LIN {X 0,Y 64.411,Z 489.736,A -85,B 0,C 180,E1 -30610.877,E2 -30610.877} C_VEL
LIN {X 0,Y 51.154,Z 493.638,A -85,B 0,C 180,E1 -30615.897,E2 -30615.897} C_VEL
LIN {X 0,Y 44.77,Z 495.003,A -85,B 0,C 180,E1 -30619.623,E2 -30619.623} C_VEL
LIN {X 0,Y 33.01,Z 496.515,A -85,B 0,C 180,E1 -30631.605,E2 -30631.605} C_VEL
LIN {X 0,Y 24.283,Z 496.546,A -85,B 0,C 180,E1 -30654.624,E2 -30654.624} C_VEL
LIN {X 0,Y 22.308,Z 495.994,A -85,B 0,C 180,E1 -30671.629,E2 -30671.629} C_VEL
LIN {X 0,Y 21.842,Z 494.93,A -85,B 0,C 180,E1 -30689.992,E2 -30689.992} C_VEL
LIN {X 0,Y 22.673,Z 492.2,A -85,B 0,C 180,E1 -30717.699,E2 -30717.699} C_VEL
LIN {X 0,Y 27.806,Z 488.413,A -85,B 0,C 180,E1 -30739.3,E2 -30739.3} C_VEL
LIN {X 0,Y 35.581,Z 483.511,A -85,B 0,C 180,E1 -30752.715,E2 -30752.715} C_VEL
LIN {X 0,Y 44.643,Z 477.362,A -85,B 0,C 180,E1 -30760.815,E2 -30760.815} C_VEL
LIN {X 0,Y 54.307,Z 469.729,A -85,B 0,C 180,E1 -30766.054,E2 -30766.054} C_VEL
LIN {X 0,Y 62.602,Z 461.942,A -85,B 0,C 180,E1 -30769.19,E2 -30769.19} C_VEL
LIN {X 0,Y 71.072,Z 452.525,A -85,B 0,C 180,E1 -30771.416,E2 -30771.416} C_VEL
LIN {X 0,Y 78.787,Z 442.074,A -85,B 0,C 180,E1 -30772.895,E2 -30772.895} C_VEL
LIN {X 0,Y 85.688,Z 430.488,A -85,B 0,C 180,E1 -30773.94,E2 -30773.94} C_VEL
LIN {X 0,Y 91.281,Z 418.187,A -85,B 0,C 180,E1 -30774.899,E2 -30774.899} C_VEL
LIN {X 0,Y 95.798,Z 404.539,A -85,B 0,C 180,E1 -30775.577,E2 -30775.577} C_VEL
LIN {X 0,Y 98.056,Z 394.55,A -85,B 0,C 180,E1 -30776.019,E2 -30776.019} C_VEL
LIN {X 0,Y 99.588,Z 382.636,A -85,B 0,C 180,E1 -30777.143,E2 -30777.143} C_VEL
LIN {X 0,Y 99.215,Z 380.276,A -85,B 0,C 180,E1 -30780.904,E2 -30780.904} C_VEL
LIN {X 0,Y 99.074,Z 379.59,A -85,B 0,C 180,E1 -30784.069,E2 -30784.069} C_VEL
LIN {X 0,Y 99.228,Z 380.869,A -85,B 0,C 180,E1 -30789.529,E2 -30789.529} C_VEL
LIN {X 0,Y 99.747,Z 383.531,A -85,B 0,C 180,E1 -30793.797,E2 -30793.797} C_VEL
LIN {X 0,Y 97.367,Z 397.045,A -85,B 0,C 180,E1 -30794.611,E2 -30794.611} C_VEL
LIN {X 0,Y 93.817,Z 409.498,A -85,B 0,C 180,E1 -30795.532,E2 -30795.532} C_VEL
LIN {X 0,Y 88.903,Z 421.701,A -85,B 0,C 180,E1 -30796.731,E2 -30796.731} C_VEL
LIN {X 0,Y 82.394,Z 434,A -85,B 0,C 180,E1 -30798.4,E2 -30798.4} C_VEL
LIN {X 0,Y 75.011,Z 444.958,A -85,B 0,C 180,E1 -30800.468,E2 -30800.468} C_VEL
LIN {X 0,Y 66.865,Z 454.739,A -85,B 0,C 180,E1 -30803.129,E2 -30803.129} C_VEL
LIN {X 0,Y 57.311,Z 464.214,A -85,B 0,C 180,E1 -30807.253,E2 -30807.253} C_VEL
LIN {X 0,Y 51.041,Z 469.447,A -85,B 0,C 180,E1 -30810.706,E2 -30810.706} C_VEL
LIN {X 0,Y 46.551,Z 472.773,A -85,B 0,C 180,E1 -30812.993,E2 -30812.993} C_VEL
LIN {X 0,Y 38.26,Z 477.884,A -85,B 0,C 180,E1 -30815.633,E2 -30815.633} C_VEL
LIN {X 0,Y 29.677,Z 482.288,A -85,B 0,C 180,E1 -30819.804,E2 -30819.804} C_VEL
LIN {X 0,Y 24.982,Z 484.511,A -85,B 0,C 180,E1 -30825.843,E2 -30825.843} C_VEL
LIN {X 0,Y 18.331,Z 488.004,A -85,B 0,C 180,E1 -30847.467,E2 -30847.467} C_VEL
LIN {X 0,Y 16.306,Z 489.794,A -85,B 0,C 180,E1 -30870.01,E2 -30870.01} C_VEL
LIN {X 0,Y 17.09,Z 491.165,A -85,B 0,C 180,E1 -30894.293,E2 -30894.293} C_VEL
LIN {X 0,Y 25.119,Z 492.78,A -85,B 0,C 180,E1 -30927.083,E2 -30927.083} C_VEL
LIN {X 0,Y 36.936,Z 492.769,A -85,B 0,C 180,E1 -30942.069,E2 -30942.069} C_VEL
LIN {X 0,Y 49.983,Z 491.209,A -85,B 0,C 180,E1 -30949.828,E2 -30949.828} C_VEL
LIN {X 0,Y 59.176,Z 489.158,A -85,B 0,C 180,E1 -30953.178,E2 -30953.178} C_VEL
LIN {X 0,Y 70.438,Z 485.63,A -85,B 0,C 180,E1 -30956.175,E2 -30956.175} C_VEL
LIN {X 0,Y 80.86,Z 481.242,A -85,B 0,C 180,E1 -30958.277,E2 -30958.277} C_VEL
LIN {X 0,Y 91.622,Z 475.439,A -85,B 0,C 180,E1 -30959.999,E2 -30959.999} C_VEL
LIN {X 0,Y 96.335,Z 472.448,A -85,B 0,C 180,E1 -30960.646,E2 -30960.646} C_VEL
LIN {X 0,Y 94.746,Z 473.589,A -85,B 0,C 180,E1 -30961.156,E2 -30961.156} C_VEL
LIN {X 0,Y 84.382,Z 479.86,A -85,B 0,C 180,E1 -30961.876,E2 -30961.876} C_VEL
LIN {X 0,Y 73.893,Z 484.988,A -85,B 0,C 180,E1 -30962.944,E2 -30962.944} C_VEL
LIN {X 0,Y 63.452,Z 489.025,A -85,B 0,C 180,E1 -30964.536,E2 -30964.536} C_VEL
LIN {X 0,Y 49.676,Z 492.881,A -85,B 0,C 180,E1 -30967.955,E2 -30967.955} C_VEL
LIN {X 0,Y 42.902,Z 494.21,A -85,B 0,C 180,E1 -30970.597,E2 -30970.597} C_VEL
LIN {X 0,Y 29.89,Z 495.665,A -85,B 0,C 180,E1 -30979.851,E2 -30979.851} C_VEL
LIN {X 0,Y 18.921,Z 495.653,A -85,B 0,C 180,E1 -31002.013,E2 -31002.013} C_VEL
LIN {X 0,Y 15.598,Z 495.019,A -85,B 0,C 180,E1 -31024.295,E2 -31024.295} C_VEL
LIN {X 0,Y 14.701,Z 493.969,A -85,B 0,C 180,E1 -31049.989,E2 -31049.989} C_VEL
LIN {X 0,Y 16.651,Z 491.185,A -85,B 0,C 180,E1 -31089.266,E2 -31089.266} C_VEL
LIN {X 0,Y 23.762,Z 487.35,A -85,B 0,C 180,E1 -31112.516,E2 -31112.516} C_VEL
LIN {X 0,Y 32.915,Z 482.393,A -85,B 0,C 180,E1 -31123.891,E2 -31123.891} C_VEL
LIN {X 0,Y 44.264,Z 475.215,A -85,B 0,C 180,E1 -31130.522,E2 -31130.522} C_VEL
LIN {X 0,Y 54.753,Z 467.007,A -85,B 0,C 180,E1 -31134.1,E2 -31134.1} C_VEL
LIN {X 0,Y 63.401,Z 458.843,A -85,B 0,C 180,E1 -31136.015,E2 -31136.015} C_VEL
LIN {X 0,Y 72.108,Z 448.91,A -85,B 0,C 180,E1 -31137.379,E2 -31137.379} C_VEL
LIN {X 0,Y 79.974,Z 437.823,A -85,B 0,C 180,E1 -31138.29,E2 -31138.29} C_VEL
LIN {X 0,Y 86.106,Z 426.967,A -85,B 0,C 180,E1 -31138.826,E2 -31138.826} C_VEL
LIN {X 0,Y 91.363,Z 414.899,A -85,B 0,C 180,E1 -31139.454,E2 -31139.454} C_VEL
LIN {X 0,Y 95.513,Z 401.939,A -85,B 0,C 180,E1 -31139.843,E2 -31139.843} C_VEL
LIN {X 0,Y 97.088,Z 394.945,A -85,B 0,C 180,E1 -31140.138,E2 -31140.138} C_VEL
LIN {X 0,Y 98.245,Z 387.692,A -85,B 0,C 180,E1 -31140.889,E2 -31140.889} C_VEL
LIN {X 0,Y 98.179,Z 386.794,A -85,B 0,C 180,E1 -31143.078,E2 -31143.078} C_VEL
LIN {X 0,Y 98.117,Z 386.905,A -85,B 0,C 180,E1 -31145.78,E2 -31145.78} C_VEL
LIN {X 0,Y 98.168,Z 387.884,A -85,B 0,C 180,E1 -31148.759,E2 -31148.759} C_VEL
LIN {X 0,Y 98.217,Z 388.502,A -85,B 0,C 180,E1 -31149.881,E2 -31149.881} C_VEL
LIN {X 0,Y 95.367,Z 401.671,A -85,B 0,C 180,E1 -31150.723,E2 -31150.723} C_VEL
LIN {X 0,Y 91.031,Z 414.726,A -85,B 0,C 180,E1 -31151.582,E2 -31151.582} C_VEL
LIN {X 0,Y 85.522,Z 426.812,A -85,B 0,C 180,E1 -31152.629,E2 -31152.629} C_VEL
LIN {X 0,Y 78.767,Z 438.222,A -85,B 0,C 180,E1 -31154.007,E2 -31154.007} C_VEL
LIN {X 0,Y 71.163,Z 448.53,A -85,B 0,C 180,E1 -31155.67,E2 -31155.67} C_VEL
LIN {X 0,Y 62.756,Z 457.831,A -85,B 0,C 180,E1 -31157.854,E2 -31157.854} C_VEL
LIN {X 0,Y 52.775,Z 466.807,A -85,B 0,C 180,E1 -31161.233,E2 -31161.233} C_VEL
LIN {X 0,Y 43.034,Z 474.039,A -85,B 0,C 180,E1 -31166.088,E2 -31166.088} C_VEL
LIN {X 0,Y 33.729,Z 479.835,A -85,B 0,C 180,E1 -31173.555,E2 -31173.555} C_VEL
LIN {X 0,Y 24.982,Z 484.511,A -85,B 0,C 180,E1 -31185.843,E2 -31185.843} C_VEL
LIN {X 0,Y 20.607,Z 486.568,A -85,B 0,C 180,E1 -31194.559,E2 -31194.559} C_VEL
LIN {X 0,Y 13.507,Z 489.493,A -85,B 0,C 180,E1 -31216.216,E2 -31216.216} C_VEL
LIN {X 0,Y 10.661,Z 491.408,A -85,B 0,C 180,E1 -31251.051,E2 -31251.051} C_VEL
LIN {X 0,Y 13.106,Z 492.624,A -85,B 0,C 180,E1 -31282.171,E2 -31282.171} C_VEL
LIN {X 0,Y 13.792,Z 492.698,A -85,B 0,C 180,E1 -31285.129,E2 -31285.129} C_VEL
LIN {X 0,Y 22.075,Z 493.659,A -85,B 0,C 180,E1 -31302.791,E2 -31302.791} C_VEL
LIN {X 0,Y 35.396,Z 493.594,A -85,B 0,C 180,E1 -31313.136,E2 -31313.136} C_VEL
LIN {X 0,Y 42.274,Z 492.99,A -85,B 0,C 180,E1 -31315.973,E2 -31315.973} C_VEL
LIN {X 0,Y 49.227,Z 491.971,A -85,B 0,C 180,E1 -31318.023,E2 -31318.023} C_VEL
LIN {X 0,Y 49.198,Z 492.124,A -85,B 0,C 180,E1 -31319.698,E2 -31319.698} C_VEL
LIN {X 0,Y 42.177,Z 493.408,A -85,B 0,C 180,E1 -31321.021,E2 -31321.021} C_VEL
LIN {X 0,Y 28.274,Z 494.816,A -85,B 0,C 180,E1 -31326.09,E2 -31326.09} C_VEL
LIN {X 0,Y 15.103,Z 494.749,A -85,B 0,C 180,E1 -31341.428,E2 -31341.428} C_VEL
LIN {X 0,Y 9.366,Z 494.009,A -85,B 0,C 180,E1 -31368.612,E2 -31368.612} C_VEL
LIN {X 0,Y 7.562,Z 493.009,A -85,B 0,C 180,E1 -31409.978,E2 -31409.978} C_VEL
LIN {X 0,Y 11.976,Z 490.169,A -85,B 0,C 180,E1 -31471.639,E2 -31471.639} C_VEL
LIN {X 0,Y 21.417,Z 486.286,A -85,B 0,C 180,E1 -31489.831,E2 -31489.831} C_VEL
LIN {X 0,Y 31.683,Z 481.277,A -85,B 0,C 180,E1 -31496.443,E2 -31496.443} C_VEL
LIN {X 0,Y 42.166,Z 475.016,A -85,B 0,C 180,E1 -31499.507,E2 -31499.507} C_VEL
LIN {X 0,Y 52.721,Z 467.233,A -85,B 0,C 180,E1 -31501.386,E2 -31501.386} C_VEL
LIN {X 0,Y 61.542,Z 459.291,A -85,B 0,C 180,E1 -31502.341,E2 -31502.341} C_VEL
LIN {X 0,Y 70.371,Z 449.607,A -85,B 0,C 180,E1 -31502.993,E2 -31502.993} C_VEL
LIN {X 0,Y 78.31,Z 438.92,A -85,B 0,C 180,E1 -31503.275,E2 -31503.275} C_VEL
LIN {X 0,Y 84.489,Z 428.581,A -85,B 0,C 180,E1 -31503.505,E2 -31503.505} C_VEL
LIN {X 0,Y 89.803,Z 417.326,A -85,B 0,C 180,E1 -31503.834,E2 -31503.834} C_VEL
LIN {X 0,Y 94.327,Z 404.368,A -85,B 0,C 180,E1 -31504.081,E2 -31504.081} C_VEL
LIN {X 0,Y 96.651,Z 395.221,A -85,B 0,C 180,E1 -31504.344,E2 -31504.344} C_VEL
LIN {X 0,Y 96.937,Z 393.716,A -85,B 0,C 180,E1 -31504.573,E2 -31504.573} C_VEL
LIN {X 0,Y 96.848,Z 394.168,A -85,B 0,C 180,E1 -31506.028,E2 -31506.028} C_VEL
LIN {X 0,Y 93.844,Z 405.878,A -85,B 0,C 180,E1 -31506.633,E2 -31506.633} C_VEL
LIN {X 0,Y 89.08,Z 418.671,A -85,B 0,C 180,E1 -31507.336,E2 -31507.336} C_VEL
LIN {X 0,Y 83.411,Z 430.103,A -85,B 0,C 180,E1 -31508.125,E2 -31508.125} C_VEL
LIN {X 0,Y 76.506,Z 441.074,A -85,B 0,C 180,E1 -31509.086,E2 -31509.086} C_VEL
LIN {X 0,Y 69.595,Z 449.982,A -85,B 0,C 180,E1 -31510.093,E2 -31510.093} C_VEL
LIN {X 0,Y 60.969,Z 459.14,A -85,B 0,C 180,E1 -31511.555,E2 -31511.555} C_VEL
LIN {X 0,Y 50.651,Z 468.041,A -85,B 0,C 180,E1 -31513.785,E2 -31513.785} C_VEL
LIN {X 0,Y 40.435,Z 475.205,A -85,B 0,C 180,E1 -31517.085,E2 -31517.085} C_VEL
LIN {X 0,Y 30.402,Z 480.936,A -85,B 0,C 180,E1 -31522.399,E2 -31522.399} C_VEL
LIN {X 0,Y 20.659,Z 485.495,A -85,B 0,C 180,E1 -31531.753,E2 -31531.753} C_VEL
LIN {X 0,Y 12.1,Z 489.003,A -85,B 0,C 180,E1 -31554.508,E2 -31554.508} C_VEL
LIN {X 0,Y 9.228,Z 490.75,A -85,B 0,C 180,E1 -31590.018,E2 -31590.018} C_VEL
LIN {X 0,Y 13.792,Z 492.698,A -85,B 0,C 180,E1 -31645.129,E2 -31645.129} C_VEL
LIN {X 0,Y 13.353,Z 492.858,A -85,B 0,C 180,E1 -31648.212,E2 -31648.212} C_VEL
LIN {X 0,Y 10.848,Z 492.885,A -85,B 0,C 180,E1 -31651.01,E2 -31651.01} C_VEL
LIN {X 0,Y 7.416,Z 492.641,A -85,B 0,C 180,E1 -31650.293,E2 -31650.293} C_VEL
LIN {X 0,Y 2.4,Z 491.412,A -85,B 0,C 180,E1 -31531.268,E2 -31531.268} C_VEL
LIN {X 0,Y 6.851,Z 490.301,A -85,B 0,C 180,E1 -31507.657,E2 -31507.657} C_VEL
LIN {X 0,Y 8.723,Z 489.747,A -85,B 0,C 180,E1 -31507.488,E2 -31507.488} C_VEL
LIN {X 0,Y 21.355,Z 485.22,A -85,B 0,C 180,E1 -31509.202,E2 -31509.202} C_VEL
LIN {X 0,Y 21.468,Z 485.124,A -85,B 0,C 180,E1 -31510.906,E2 -31510.906} C_VEL
LIN {X 0,Y 10.993,Z 488.924,A -85,B 0,C 180,E1 -31516.536,E2 -31516.536} C_VEL
LIN {X 0,Y 2.151,Z 491.702,A -85,B 0,C 180,E1 -31590.078,E2 -31590.078} C_VEL
LIN {X 0,Y 7.165,Z 493.032,A -85,B 0,C 180,E1 -31668.908,E2 -31668.908} C_VEL
LIN {X 0,Y 7.036,Z 493.179,A -85,B 0,C 180,E1 -31677.875,E2 -31677.875} C_VEL
LIN {X 0,Y 0.427,Z 492.049,A -85,B 0,C 180,E1 -31769.605,E2 -31769.605} C_VEL
LIN {X 0,Y 8.723,Z 489.747,A -85,B 0,C 180,E1 -31867.488,E2 -31867.488} C_VEL
LIN {X 0,Y 11.308,Z 491.658,A -85,B 0,C 180,E1 -31868.242,E2 -31868.242} C_VEL
LIN {X 0,Y 11.308,Z 600,A -85,B 0,C 180,E1 -31868.242,E2 -31868.242} C_VEL
LIN {X 0,Y 11.308,Z 600,A -85,B 0,C 180,E1 -31868.242,E2 -31868.242}

QRS_NEXT_CUT()

QRS_NEXT()
QRS_HOME()

END
